(*	Struktura zawierające dane tylko tego elementu	*)
TYPE ST_Component_HMI_Link EXTENDS ST_BaseComponent_HMI_Link :
STRUCT
	stComponent			: ST_Component_HMI;

END_STRUCT
END_TYPE

(* stored: Version 1.1.0.1, ProductVersion 3.1.4024.15
   DUT ST_Component_HMI_Link: Id {216acca6-72b9-42d5-bfc6-2be5c27a09ff} *)
